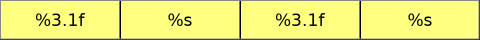
VISUALIZATION VISU_CONFIG_LIGNE_GAZ_SURV_MFC_MKS  // 480x40
VAR_IN_OUT
	m_Input_MASSFLOW:		BLOCK_MFC_MKS_NoCoE;
END_VAR
    Rectangle (0,0 120x40), "%3.1f", text variable: m_Input_MASSFLOW.VAR_ALM_SURV.OFFSET, input disabled if: NOT Global_Variables.PRG_USER.ACTU_USER.CONF_MACHINE
        OnMouseDown: write the text variable via Edit
    Rectangle (240,0 120x40), "%3.1f", text variable: m_Input_MASSFLOW.VAR_DEF_SURV.offset, input disabled if: NOT Global_Variables.PRG_USER.ACTU_USER.CONF_MACHINE
        OnMouseDown: write the text variable via VisuDialogs.Numpad
    Rectangle (120,0 120x40), "%s", text variable: m_Input_MASSFLOW.ALM_SURV.delay, input disabled if: NOT Global_Variables.PRG_USER.ACTU_USER.CONF_MACHINE
        OnMouseDown: write the text variable via VisuDialogs.Keypad
    Rectangle (360,0 120x40), "%s", text variable: m_Input_MASSFLOW.DEF_SURV.DELAY, input disabled if: NOT Global_Variables.PRG_USER.ACTU_USER.CONF_MACHINE
        OnMouseDown: write the text variable via VisuDialogs.Keypad
END_VISUALIZATION

(* stored: Version 1.1.0.1, ProductVersion 3.1.4024.6
   Visu VISU_CONFIG_LIGNE_GAZ_SURV_MFC_MKS: Id {f7ab6c72-e8bb-43f2-afb6-7be734d96dda} *)
